// TIA Portal project "Esvetovaya" (V17)

(* hardware
DEVICE "S7-1200 station_1"  S7-1200 Station
   slot 0: "Rack_0"  S7-1200 Rack  Rack  V1.0
   slot 1: "PLC_1"  CPU 1214C AC/DC/Rly  6ES7 214-1BG40-0XB0  V4.5
*)

// ===== PLC "PLC_1"  CPU 1214C AC/DC/Rly =====

VAR_GLOBAL   // PLC tag table "TDB_Output_Q"
   "Q0.0_Lamp_Auto" AT %Q0.0 : Bool;   // Luces de modo automatico
   "Q0.1_Lamp_Manu" AT %Q0.1 : Bool;   // Luces de modo manual
   "Q0.2_Relay_ON" AT %Q0.2 : Bool;   // SAlida del soplador
   "Q0.3_Relay_ON" AT %Q0.3 : Bool;   // SAlida del soplador
   "Q0.4_Relay_ON" AT %Q0.4 : Bool;   // Salida de calefaccion
   "Q0.5_Relay_On" AT %Q0.5 : Bool;   // Salida de nebulizacion
   "Q1.0_Lamp_Auto_Running" AT %Q1.0 : Bool;   // Luces de modo de funcionamiento automatico
END_VAR

VAR_GLOBAL   // PLC tag table "TDB_Input_I"
   "I_Btt_Auto_Q0" AT %I0.0 : Bool;   // Modo de operacion Automatica
   "I_Btt_Manu_Q1" AT %I0.1 : Bool;   // Modo de operacion Manual
   "I_Btt_Start_Q2" AT %I0.2 : Bool;   // Interruptor de parada de funcionamiento del soplador
   "I_Btt___Off_Q2" AT %I0.3 : Bool;   // interruptor vegetariano deja de calentar
   "I_Btt_Start_Q3" AT %I0.4 : Bool;   // interruptor de funcionamiento detener nebulizacion
   "I_Btt___Off_Q3" AT %I0.5 : Bool;   // boton pulsador se ejecuta automaticamente
   "I_Btt_Start_Q4" AT %I0.6 : Bool;   // pulsador de parada automatica
   "Sensor_PT100" AT %IW64 : Int;   // sensor de temperatura
END_VAR

VAR_GLOBAL   // PLC tag table "M_Variables"
   "M_Btt_auto_Q0" AT %M0.0 : Bool;   // Memoria_Modo de operacion Automatica
   "M_Btt_Manu_Q1" AT %M0.1 : Bool;   // Memoria_Modo de operacion Manual
   "M_AUTO" AT %M0.2 : Bool;
   "M_MANUAL" AT %M0.3 : Bool;
   "M_Btt_Auto_On" AT %M0.4 : Bool;   // Memoria_boton pulsador se ejecuta automaticamente
   "M_Btt_Auto_Off" AT %M0.5 : Bool;   // Memoria_pulsador de parada automatica
   "ReStart" AT %M1.0 : Bool;
   "Bucle_Amarillo" AT %M1.1 : Bool;
   "Bucle_Rojo" AT %M1.3 : Bool;
   "M_SinEntender" AT %M1.4 : Bool;
   "M_Simulation" AT %M1.5 : Bool;   // Enciende la funciona de simulacion
   "Mtime_Lectura_Sensor" AT %M2.0 : Bool;
   "MQ2_Manu_Start" AT %M3.0 : Bool;   // Nebulizacion manual de modo intermedio
   "MQ2_Manu_Stop" AT %M3.1 : Bool;
   "MQ3_Manu_Start" AT %M3.2 : Bool;   // Soplador manual de modo intermedio
   "MQ3_Manu_Stop" AT %M3.3 : Bool;   // Calefaccion Manual de modo intermedio
   "MQ2_Auto_Start1" AT %M4.0 : Bool;   // Calentamiento Automatico en modo intermedio
   "MQ2_Auto_Start2" AT %M4.1 : Bool;   // Calentamiento Automatico en modo intermedio
   "MQ2_Auto_Start3" AT %M4.2 : Bool;   // Calentamiento Automatico en modo intermedio
   "MQ2_Auto_Stop" AT %M4.3 : Bool;
   "MQ2_Remote_Start" AT %M5.0 : Bool;   // Memoria_Interruptor de parada de funcionamiento del soplador
   "MQ3_Remote_Start" AT %M5.1 : Bool;   // Memoria_interruptor de funcionamiento detener nebulizacion
   "MQ2_Remote_Stop" AT %M5.2 : Bool;
   "MQ3_Remote_Stop" AT %M5.3 : Bool;
   "foco" AT %M6.0 : Bool;
END_VAR

DATA_BLOCK "DB_Sensors"   // DB1
{ S7_Optimized_Access := 'FALSE' }
VERSION : 0.1
   VAR
      Data_Norm_PT100 : Real;
      Data_Redondeo_PT100 : Real;
      Data_Scalado_PT100 : Real;
      Data_Evaluation_TempPT100 : Real := 25.0;
      Temp_Min : Real := 20.0;
      Temp_Max : Real := 27.0;
   END_VAR
BEGIN
END_DATA_BLOCK

DATA_BLOCK "DB_Clock"   // DB2
{ S7_Optimized_Access := 'TRUE' }
VERSION : 0.1
   VAR
      Fecha_hora_1_sistema : DTL := DTL#1970-01-01-00:00:00;
      Fecha_hora_2_sistema : DTL := DTL#1970-01-01-00:00:00;
      Fecha_hora_1_local : DTL := DTL#1970-01-01-00:00:00;
      Fecha_hora_2_local : DTL := DTL#1970-01-01-00:00:00;
      Ret_val_sistema_1 : Word := 16#0;
      Ret_val_sistema_2 : Word := 16#0;
      Ret_val_local_1 : Word := 16#0;
      Ret_val_local_2 : Word := 16#0;
      Hora_sistema_1 : Time_Of_Day := TOD#00:00:00;
      Hora_sistema_2 : Time_Of_Day := TOD#00:00:00;
      Hora_local_1 : Time_Of_Day := TOD#00:00:00;
      Hora_local_2 : Time_Of_Day := TOD#00:00:00;
      Hora_Q2_inicio_1 : Time_Of_Day := TOD#00:00:00;
      Hora_Q2_inicio_2 : Time_Of_Day := TOD#00:00:00;
      Hora_Q2_inicio_3 : Time_Of_Day := TOD#00:00:00;
      Hora_Q3_inicio_1 : Time_Of_Day := TOD#00:00:00;
      Hora_Q3_inicio_2 : Time_Of_Day := TOD#00:00:00;
      Hora_Q3_inicio_3 : Time_Of_Day := TOD#00:00:00;
      Hora_Q2_fin_1 : Time_Of_Day := TOD#00:00:00;
      Hora_Q2_fin_2 : Time_Of_Day := TOD#00:00:00;
      Hora_Q2_fin_3 : Time_Of_Day := TOD#00:00:00;
      Hora_Q3_fin_1 : Time_Of_Day := TOD#00:00:00;
      Hora_Q3_fin_2 : Time_Of_Day := TOD#00:00:00;
      Hora_Q3_fin_3 : Time_Of_Day := TOD#00:00:00;
      Hora_Start_ARR_Q2_1 : Array[1..7] of Time_Of_Day;
      Hora_Start_ARR_Q2_2 : Array[1..7] of Time_Of_Day;
      Hora_Start_ARR_Q2_3 : Array[1..7] of Time_Of_Day;
      Hora_Start_ARR_Q3_1 : Array[1..7] of Time_Of_Day;
      Hora_Start_ARR_Q3_2 : Array[1..7] of Time_Of_Day;
      Hora_Start_ARR_Q3_3 : Array[1..7] of Time_Of_Day;
      Hora_End_ARR_Q2_1 : Array[1..7] of Time_Of_Day;
      Hora_End_ARR_Q2_2 : Array[1..7] of Time_Of_Day;
      Hora_End_ARR_Q2_3 : Array[1..7] of Time_Of_Day;
      Hora_End_ARR_Q3_1 : Array[1..7] of Time_Of_Day;
      Hora_End_ARR_Q3_2 : Array[1..7] of Time_Of_Day;
      Hora_End_ARR_Q3_3 : Array[1..7] of Time_Of_Day;
   END_VAR
BEGIN
   Hora_Start_ARR_Q2_1[1] := TOD#06:00:00;
   Hora_Start_ARR_Q2_1[2] := TOD#06:00:00;
   Hora_Start_ARR_Q2_1[3] := TOD#06:00:00;
   Hora_Start_ARR_Q2_1[4] := TOD#06:00:00;
   Hora_Start_ARR_Q2_1[5] := TOD#06:00:00;
   Hora_Start_ARR_Q2_1[6] := TOD#06:00:00;
   Hora_Start_ARR_Q2_1[7] := TOD#06:00:00;
   Hora_End_ARR_Q2_1[1] := TOD#20:00:00;
   Hora_End_ARR_Q2_1[2] := TOD#20:00:00;
   Hora_End_ARR_Q2_1[3] := TOD#20:00:00;
   Hora_End_ARR_Q2_1[4] := TOD#20:00:00;
   Hora_End_ARR_Q2_1[5] := TOD#20:00:00;
   Hora_End_ARR_Q2_1[6] := TOD#20:00:00;
   Hora_End_ARR_Q2_1[7] := TOD#20:00:00;
   Hora_Start_ARR_Q2_2[1] := TOD#06:00:00;
   Hora_Start_ARR_Q2_2[2] := TOD#06:00:00;
   Hora_Start_ARR_Q2_2[3] := TOD#06:00:00;
   Hora_Start_ARR_Q2_2[4] := TOD#06:00:00;
   Hora_Start_ARR_Q2_2[5] := TOD#06:00:00;
   Hora_Start_ARR_Q2_2[6] := TOD#06:00:00;
   Hora_Start_ARR_Q2_2[7] := TOD#06:00:00;
   Hora_Start_ARR_Q2_3[1] := TOD#06:00:00;
   Hora_Start_ARR_Q2_3[2] := TOD#06:00:00;
   Hora_Start_ARR_Q2_3[3] := TOD#06:00:00;
   Hora_Start_ARR_Q2_3[4] := TOD#06:00:00;
   Hora_Start_ARR_Q2_3[5] := TOD#06:00:00;
   Hora_Start_ARR_Q2_3[6] := TOD#06:00:00;
   Hora_Start_ARR_Q2_3[7] := TOD#06:00:00;
   Hora_Start_ARR_Q3_1[1] := TOD#06:00:00;
   Hora_Start_ARR_Q3_1[2] := TOD#06:00:00;
   Hora_Start_ARR_Q3_1[3] := TOD#06:00:00;
   Hora_Start_ARR_Q3_1[4] := TOD#06:00:00;
   Hora_Start_ARR_Q3_1[5] := TOD#06:00:00;
   Hora_Start_ARR_Q3_1[6] := TOD#06:00:00;
   Hora_Start_ARR_Q3_1[7] := TOD#06:00:00;
   Hora_Start_ARR_Q3_2[1] := TOD#06:00:00;
   Hora_Start_ARR_Q3_2[2] := TOD#06:00:00;
   Hora_Start_ARR_Q3_2[3] := TOD#06:00:00;
   Hora_Start_ARR_Q3_2[4] := TOD#06:00:00;
   Hora_Start_ARR_Q3_2[5] := TOD#06:00:00;
   Hora_Start_ARR_Q3_2[6] := TOD#06:00:00;
   Hora_Start_ARR_Q3_2[7] := TOD#06:00:00;
   Hora_Start_ARR_Q3_3[1] := TOD#06:00:00;
   Hora_Start_ARR_Q3_3[2] := TOD#06:00:00;
   Hora_Start_ARR_Q3_3[3] := TOD#06:00:00;
   Hora_Start_ARR_Q3_3[4] := TOD#06:00:00;
   Hora_Start_ARR_Q3_3[5] := TOD#06:00:00;
   Hora_Start_ARR_Q3_3[6] := TOD#06:00:00;
   Hora_Start_ARR_Q3_3[7] := TOD#06:00:00;
   Hora_End_ARR_Q2_2[1] := TOD#20:00:00;
   Hora_End_ARR_Q2_2[2] := TOD#20:00:00;
   Hora_End_ARR_Q2_2[3] := TOD#20:00:00;
   Hora_End_ARR_Q2_2[4] := TOD#20:00:00;
   Hora_End_ARR_Q2_2[5] := TOD#20:00:00;
   Hora_End_ARR_Q2_2[6] := TOD#20:00:00;
   Hora_End_ARR_Q2_2[7] := TOD#20:00:00;
   Hora_End_ARR_Q2_3[1] := TOD#20:00:00;
   Hora_End_ARR_Q2_3[2] := TOD#20:00:00;
   Hora_End_ARR_Q2_3[3] := TOD#20:00:00;
   Hora_End_ARR_Q2_3[4] := TOD#20:00:00;
   Hora_End_ARR_Q2_3[5] := TOD#20:00:00;
   Hora_End_ARR_Q2_3[6] := TOD#20:00:00;
   Hora_End_ARR_Q2_3[7] := TOD#20:00:00;
   Hora_End_ARR_Q3_1[1] := TOD#20:00:00;
   Hora_End_ARR_Q3_1[2] := TOD#20:00:00;
   Hora_End_ARR_Q3_1[3] := TOD#20:00:00;
   Hora_End_ARR_Q3_1[4] := TOD#20:00:00;
   Hora_End_ARR_Q3_1[5] := TOD#20:00:00;
   Hora_End_ARR_Q3_1[6] := TOD#20:00:00;
   Hora_End_ARR_Q3_1[7] := TOD#20:00:00;
   Hora_End_ARR_Q3_2[1] := TOD#20:00:00;
   Hora_End_ARR_Q3_2[2] := TOD#20:00:00;
   Hora_End_ARR_Q3_2[3] := TOD#20:00:00;
   Hora_End_ARR_Q3_2[4] := TOD#20:00:00;
   Hora_End_ARR_Q3_2[5] := TOD#20:00:00;
   Hora_End_ARR_Q3_2[6] := TOD#20:00:00;
   Hora_End_ARR_Q3_2[7] := TOD#20:00:00;
   Hora_End_ARR_Q3_3[1] := TOD#20:00:00;
   Hora_End_ARR_Q3_3[2] := TOD#20:00:00;
   Hora_End_ARR_Q3_3[3] := TOD#20:00:00;
   Hora_End_ARR_Q3_3[4] := TOD#20:00:00;
   Hora_End_ARR_Q3_3[5] := TOD#20:00:00;
   Hora_End_ARR_Q3_3[6] := TOD#20:00:00;
   Hora_End_ARR_Q3_3[7] := TOD#20:00:00;
END_DATA_BLOCK

DATA_BLOCK "DB_Retain"   // DB3
{ S7_Optimized_Access := 'TRUE' }
VERSION : 0.1
   VAR RETAIN
      M_Btt_auto : Bool;
   END_VAR
BEGIN
END_DATA_BLOCK

DATA_BLOCK "Datos"   // DB7
{ S7_Optimized_Access := 'FALSE' }
VERSION : 0.1
   VAR
      Static_1 : Bool;
      DatoEntero : Array[0..4] of Int;
      DatoReal : Array[0..4] of Real;
      DatoWord : Array[0..4] of Word;
      DatoBooleano : Array[0..4] of Bool;
   END_VAR
BEGIN
END_DATA_BLOCK

DATA_BLOCK "DB_Input"   // DB8
{ S7_Optimized_Access := 'TRUE' }
VERSION : 0.1
   VAR
      "1" : Bool;
   END_VAR
BEGIN
END_DATA_BLOCK

// folder: System blocks/Program resources

DATA_BLOCK "IEC_Timer_0_DB"   // DB4
{ S7_Optimized_Access := 'TRUE' }
AUTHOR : Simatic
FAMILY : IEC
NAME : IEC_TMR
VERSION : 1.0
// stored: InstanceOfName IEC_TIMER
"IEC_TIMER"
BEGIN
END_DATA_BLOCK

DATA_BLOCK "IEC_Timer_0_DB_1"   // DB5
{ S7_Optimized_Access := 'TRUE' }
AUTHOR : Simatic
FAMILY : IEC
NAME : IEC_TMR
VERSION : 1.0
// stored: InstanceOfName IEC_TIMER
"IEC_TIMER"
BEGIN
END_DATA_BLOCK

DATA_BLOCK "IEC_Timer_0_DB_2"   // DB6
{ S7_Optimized_Access := 'TRUE' }
AUTHOR : Simatic
FAMILY : IEC
NAME : IEC_TMR
VERSION : 1.0
// stored: InstanceOfName IEC_TIMER
"IEC_TIMER"
BEGIN
END_DATA_BLOCK

// folder: (top level)

FUNCTION "FC_MANUAL" : Void   // FC1, LAD
{ S7_Optimized_Access := 'TRUE' }
VERSION : 0.1
BEGIN

REGION Network 1: выход Q2 - MANUAL-(ON-OFF)
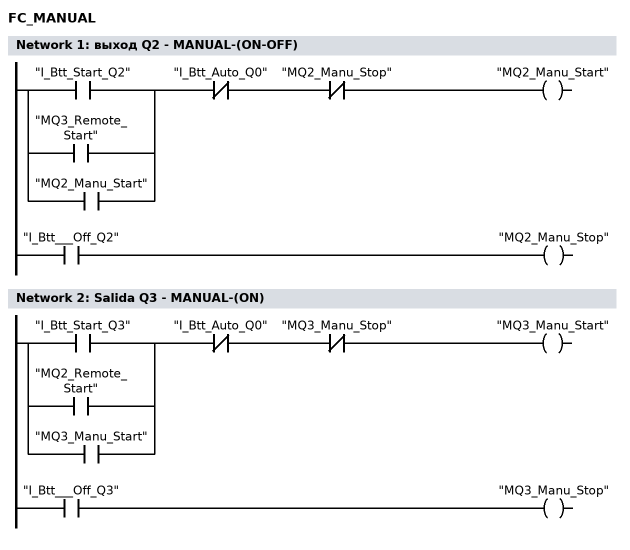
   RUNG wire#powerrail
      Contact( "I_Btt_Start_Q2" )
      wire#w1
      I_Contact( "I_Btt_Auto_Q0" )
      I_Contact( "MQ2_Manu_Stop" )
      Coil( "MQ2_Manu_Start" )
   END_RUNG
   RUNG wire#powerrail
      Contact( "MQ3_Remote_Start" )
   END_RUNG wire#w1
   RUNG wire#powerrail
      Contact( "MQ2_Manu_Start" )
   END_RUNG wire#w1
   RUNG wire#powerrail
      Contact( "I_Btt___Off_Q2" )
      Coil( "MQ2_Manu_Stop" )
   END_RUNG
   // the same network as SCL:
   "MQ2_Manu_Start" := ("I_Btt_Start_Q2" OR "MQ3_Remote_Start" OR "MQ2_Manu_Start") AND NOT "I_Btt_Auto_Q0" AND NOT "MQ2_Manu_Stop";
   "MQ2_Manu_Stop" := "I_Btt___Off_Q2";
END_REGION

REGION Network 2: Salida Q3 - MANUAL-(ON)
   RUNG wire#powerrail
      Contact( "I_Btt_Start_Q3" )
      wire#w1
      I_Contact( "I_Btt_Auto_Q0" )
      I_Contact( "MQ3_Manu_Stop" )
      Coil( "MQ3_Manu_Start" )
   END_RUNG
   RUNG wire#powerrail
      Contact( "MQ2_Remote_Start" )
   END_RUNG wire#w1
   RUNG wire#powerrail
      Contact( "MQ3_Manu_Start" )
   END_RUNG wire#w1
   RUNG wire#powerrail
      Contact( "I_Btt___Off_Q3" )
      Coil( "MQ3_Manu_Stop" )
   END_RUNG
   // the same network as SCL:
   "MQ3_Manu_Start" := ("I_Btt_Start_Q3" OR "MQ2_Remote_Start" OR "MQ3_Manu_Start") AND NOT "I_Btt_Auto_Q0" AND NOT "MQ3_Manu_Stop";
   "MQ3_Manu_Stop" := "I_Btt___Off_Q3";
END_REGION
END_FUNCTION

FUNCTION "FC_AUTO" : Void   // FC2, LAD
{ S7_Optimized_Access := 'TRUE' }
VERSION : 0.1
BEGIN

REGION Network 1: Memoria REINICIO PLC-AUTOMATICO
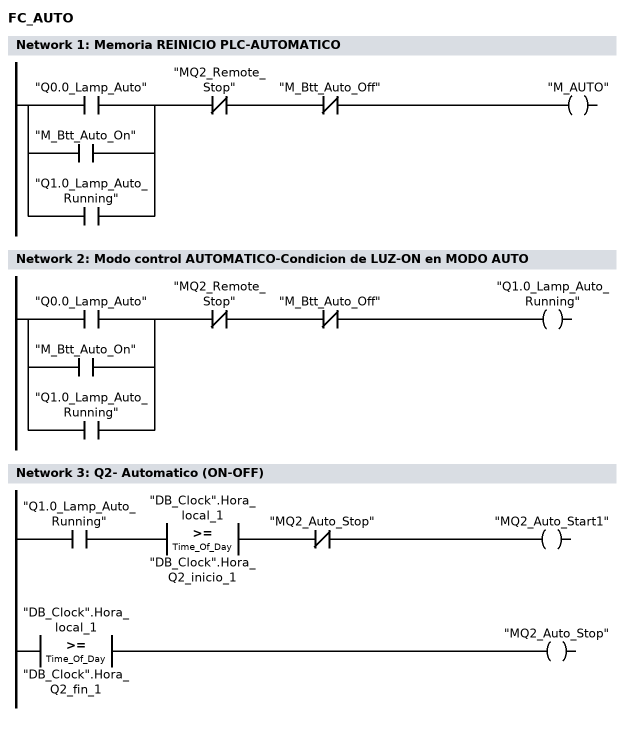
   RUNG wire#powerrail
      Contact( "Q0.0_Lamp_Auto" )
      wire#w1
      I_Contact( "MQ2_Remote_Stop" )
      I_Contact( "M_Btt_Auto_Off" )
      Coil( "M_AUTO" )
   END_RUNG
   RUNG wire#powerrail
      Contact( "M_Btt_Auto_On" )
   END_RUNG wire#w1
   RUNG wire#powerrail
      Contact( "Q1.0_Lamp_Auto_Running" )
   END_RUNG wire#w1
   // the same network as SCL:
   "M_AUTO" := ("Q0.0_Lamp_Auto" OR "M_Btt_Auto_On" OR "Q1.0_Lamp_Auto_Running") AND NOT "MQ2_Remote_Stop" AND NOT "M_Btt_Auto_Off";
END_REGION

REGION Network 2: Modo control AUTOMATICO-Condicion de LUZ-ON en MODO AUTO
   RUNG wire#powerrail
      Contact( "Q0.0_Lamp_Auto" )
      wire#w1
      I_Contact( "MQ2_Remote_Stop" )
      I_Contact( "M_Btt_Auto_Off" )
      Coil( "Q1.0_Lamp_Auto_Running" )
   END_RUNG
   RUNG wire#powerrail
      Contact( "M_Btt_Auto_On" )
   END_RUNG wire#w1
   RUNG wire#powerrail
      Contact( "Q1.0_Lamp_Auto_Running" )
   END_RUNG wire#w1
   // the same network as SCL:
   "Q1.0_Lamp_Auto_Running" := ("Q0.0_Lamp_Auto" OR "M_Btt_Auto_On" OR "Q1.0_Lamp_Auto_Running") AND NOT "MQ2_Remote_Stop" AND NOT "M_Btt_Auto_Off";
END_REGION

REGION Network 3: Q2- Automatico (ON-OFF)
   RUNG wire#powerrail
      Contact( "Q1.0_Lamp_Auto_Running" )
      { S7_Templates := "SrcType := Time_Of_Day" } GE_Contact(in1 := "DB_Clock".Hora_local_1, in2 := "DB_Clock".Hora_Q2_inicio_1)
      I_Contact( "MQ2_Auto_Stop" )
      Coil( "MQ2_Auto_Start1" )
   END_RUNG
   RUNG wire#powerrail
      { S7_Templates := "SrcType := Time_Of_Day" } GE_Contact(in1 := "DB_Clock".Hora_local_1, in2 := "DB_Clock".Hora_Q2_fin_1)
      Coil( "MQ2_Auto_Stop" )
   END_RUNG
   // the same network as SCL:
   "MQ2_Auto_Start1" := "Q1.0_Lamp_Auto_Running" AND ("DB_Clock".Hora_local_1 >= "DB_Clock".Hora_Q2_inicio_1) AND NOT "MQ2_Auto_Stop";
   "MQ2_Auto_Stop" := "DB_Clock".Hora_local_1 >= "DB_Clock".Hora_Q2_fin_1;
END_REGION
END_FUNCTION

FUNCTION "FC_OUTPUT_Q" : Void   // FC3, LAD
{ S7_Optimized_Access := 'TRUE' }
VERSION : 0.1
BEGIN

REGION Network 1: Salida Q-02 (On-Off)
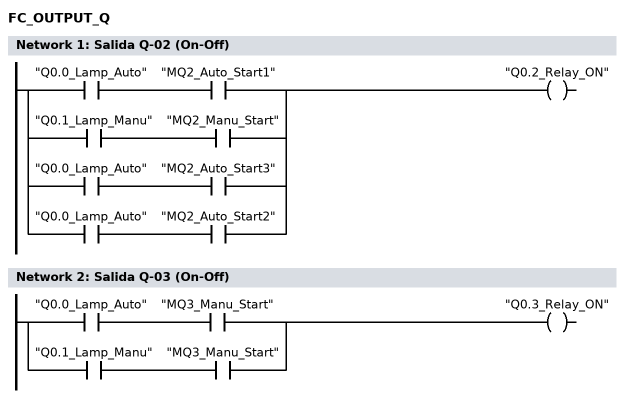
   RUNG wire#powerrail
      Contact( "Q0.0_Lamp_Auto" )
      Contact( "MQ2_Auto_Start1" )
      wire#w1
      Coil( "Q0.2_Relay_ON" )
   END_RUNG
   RUNG wire#powerrail
      Contact( "Q0.1_Lamp_Manu" )
      Contact( "MQ2_Manu_Start" )
   END_RUNG wire#w1
   RUNG wire#powerrail
      Contact( "Q0.0_Lamp_Auto" )
      Contact( "MQ2_Auto_Start3" )
   END_RUNG wire#w1
   RUNG wire#powerrail
      Contact( "Q0.0_Lamp_Auto" )
      Contact( "MQ2_Auto_Start2" )
   END_RUNG wire#w1
   // the same network as SCL:
   "Q0.2_Relay_ON" := ("Q0.0_Lamp_Auto" AND "MQ2_Auto_Start1") OR ("Q0.1_Lamp_Manu" AND "MQ2_Manu_Start") OR ("Q0.0_Lamp_Auto" AND "MQ2_Auto_Start3") OR ("Q0.0_Lamp_Auto" AND "MQ2_Auto_Start2");
END_REGION

REGION Network 2: Salida Q-03 (On-Off)
   RUNG wire#powerrail
      Contact( "Q0.0_Lamp_Auto" )
      Contact( "MQ3_Manu_Start" )
      wire#w1
      Coil( "Q0.3_Relay_ON" )
   END_RUNG
   RUNG wire#powerrail
      Contact( "Q0.1_Lamp_Manu" )
      Contact( "MQ3_Manu_Start" )
   END_RUNG wire#w1
   // the same network as SCL:
   "Q0.3_Relay_ON" := ("Q0.0_Lamp_Auto" AND "MQ3_Manu_Start") OR ("Q0.1_Lamp_Manu" AND "MQ3_Manu_Start");
END_REGION
END_FUNCTION

FUNCTION "FC_SENSORS" : Void   // FC4, LAD
{ S7_Optimized_Access := 'TRUE' }
VERSION : 0.1
BEGIN

REGION Network 1
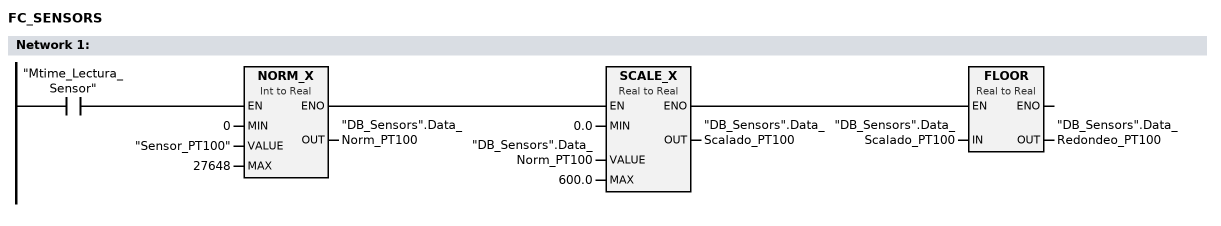
   IF "Mtime_Lectura_Sensor" THEN
       "DB_Sensors".Data_Norm_PT100 := NORM_X(MIN := 0, VALUE := "Sensor_PT100", MAX := 27648);
       "DB_Sensors".Data_Scalado_PT100 := SCALE_X(MIN := 0.0, VALUE := "DB_Sensors".Data_Norm_PT100, MAX := 600.0);
       "DB_Sensors".Data_Redondeo_PT100 := FLOOR("DB_Sensors".Data_Scalado_PT100);
   END_IF;
END_REGION
END_FUNCTION

FUNCTION "FC_CLOCK" : Void   // FC5, LAD
{ S7_Optimized_Access := 'TRUE' }
VERSION : 0.1
BEGIN

REGION Network 1: Tiempo de INTERVALO DE LECTURA FC_SENSORS
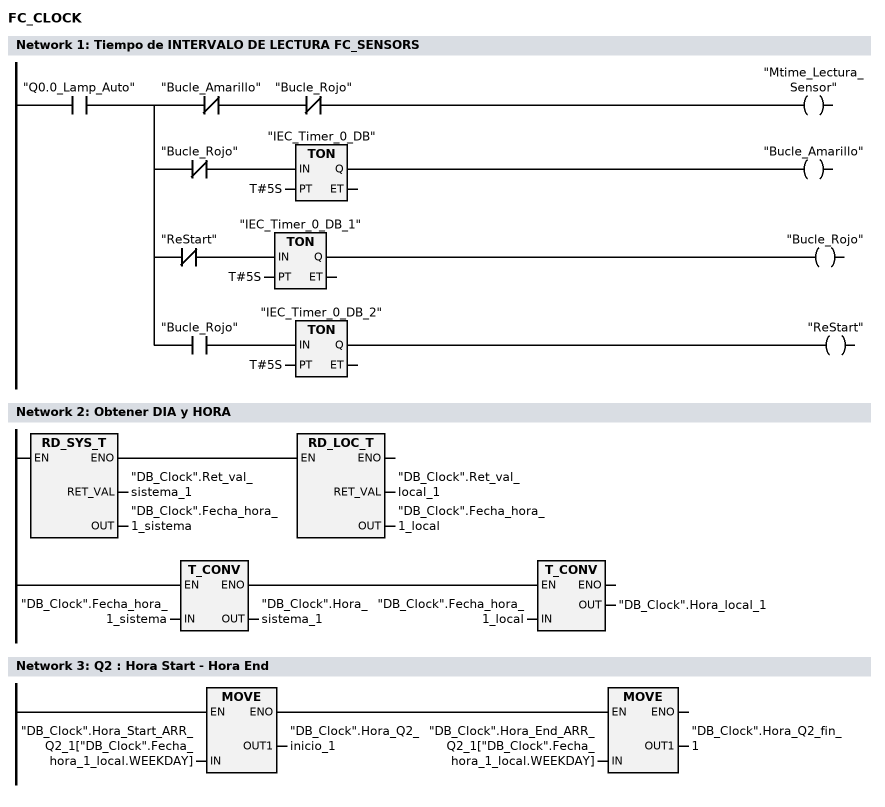
   "Mtime_Lectura_Sensor" := "Q0.0_Lamp_Auto" AND NOT "Bucle_Amarillo" AND NOT "Bucle_Rojo";
   "IEC_Timer_0_DB".TON(IN := "Q0.0_Lamp_Auto" AND NOT "Bucle_Rojo", PT := T#5S);
   "Bucle_Amarillo" := "IEC_Timer_0_DB".Q;
   "IEC_Timer_0_DB_1".TON(IN := "Q0.0_Lamp_Auto" AND NOT "ReStart", PT := T#5S);
   "Bucle_Rojo" := "IEC_Timer_0_DB_1".Q;
   "IEC_Timer_0_DB_2".TON(IN := "Q0.0_Lamp_Auto" AND "Bucle_Rojo", PT := T#5S);
   "ReStart" := "IEC_Timer_0_DB_2".Q;
END_REGION

REGION Network 2: Obtener DIA y HORA
   // ENO of a box is taken as its EN; it also drops when the box reports an error
   "DB_Clock".Ret_val_sistema_1 := RD_SYS_T(OUT => "DB_Clock".Fecha_hora_1_sistema);
   "DB_Clock".Ret_val_local_1 := RD_LOC_T(OUT => "DB_Clock".Fecha_hora_1_local);
   "DB_Clock".Hora_sistema_1 := T_CONV(IN := "DB_Clock".Fecha_hora_1_sistema);
   "DB_Clock".Hora_local_1 := T_CONV(IN := "DB_Clock".Fecha_hora_1_local);
END_REGION

REGION Network 3: Q2 : Hora Start - Hora End
   RUNG wire#powerrail
      Move(in := "DB_Clock".Hora_Start_ARR_Q2_1["DB_Clock".Fecha_hora_1_local.WEEKDAY], out1 => "DB_Clock".Hora_Q2_inicio_1)
      Move(in := "DB_Clock".Hora_End_ARR_Q2_1["DB_Clock".Fecha_hora_1_local.WEEKDAY], out1 => "DB_Clock".Hora_Q2_fin_1)
   END_RUNG
   // the same network as SCL:
   "DB_Clock".Hora_Q2_inicio_1 := "DB_Clock".Hora_Start_ARR_Q2_1["DB_Clock".Fecha_hora_1_local.WEEKDAY];
   "DB_Clock".Hora_Q2_fin_1 := "DB_Clock".Hora_End_ARR_Q2_1["DB_Clock".Fecha_hora_1_local.WEEKDAY];
END_REGION
END_FUNCTION

ORGANIZATION_BLOCK "Main"   // OB1, LAD, ProgramCycle
TITLE = "Main Program Sweep (Cycle)"
{ S7_Optimized_Access := 'TRUE' }
VERSION : 0.1
   VAR_INPUT
      Initial_Call : Bool;   // Initial call of this OB
      Remanence : Bool;   // =True, if remanent data are available
   END_VAR
   VAR_TEMP   // added for the SCL form of the ladder/FBD networks
      _w1 : Bool;
   END_VAR
BEGIN

REGION Network 1: Programa AUTOMATICO
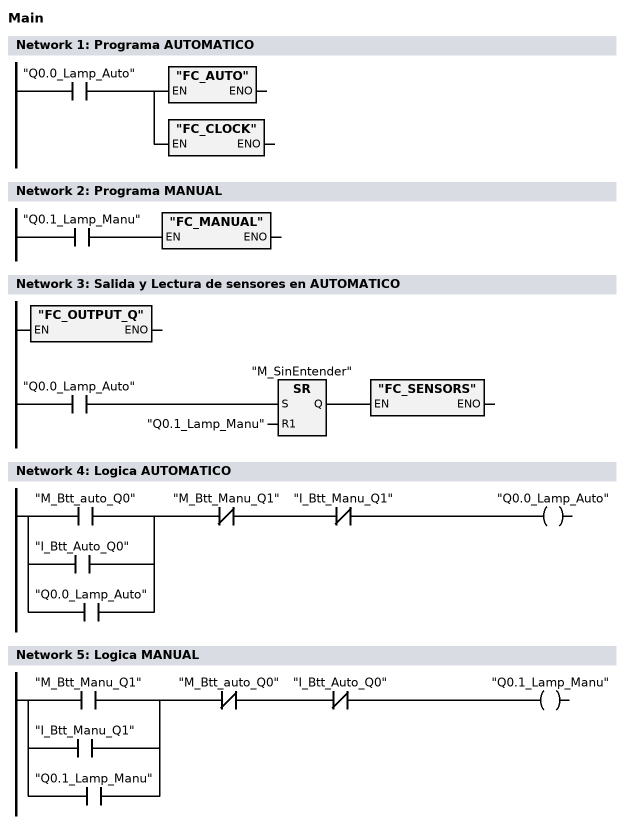
   RUNG wire#powerrail
      Contact( "Q0.0_Lamp_Auto" )
      wire#w1
      "FC_AUTO"()
   END_RUNG
   RUNG wire#w1
      "FC_CLOCK"()
   END_RUNG
   // the same network as SCL:
   #_w1 := "Q0.0_Lamp_Auto";
   IF #_w1 THEN
       "FC_AUTO"();
       "FC_CLOCK"();
   END_IF;
END_REGION

REGION Network 2: Programa MANUAL
   RUNG wire#powerrail
      Contact( "Q0.1_Lamp_Manu" )
      "FC_MANUAL"()
   END_RUNG
   // the same network as SCL:
   IF "Q0.1_Lamp_Manu" THEN "FC_MANUAL"(); END_IF;
END_REGION

REGION Network 3: Salida y Lectura de sensores en AUTOMATICO
   RUNG wire#powerrail
      "FC_OUTPUT_Q"()
   END_RUNG
   RUNG wire#powerrail
      Contact( "Q0.0_Lamp_Auto" )
      S_SR(operand := "M_SinEntender", r1 := "Q0.1_Lamp_Manu")
      "FC_SENSORS"()
   END_RUNG
   // the same network as SCL:
   "FC_OUTPUT_Q"();
   IF "Q0.0_Lamp_Auto" THEN
       "M_SinEntender" := TRUE;   // SR flip-flop
   END_IF;
   IF "Q0.1_Lamp_Manu" THEN "M_SinEntender" := FALSE; END_IF;
   IF "M_SinEntender" THEN "FC_SENSORS"(); END_IF;
END_REGION

REGION Network 4: Logica AUTOMATICO
   RUNG wire#powerrail
      Contact( "M_Btt_auto_Q0" )
      wire#w1
      I_Contact( "M_Btt_Manu_Q1" )
      I_Contact( "I_Btt_Manu_Q1" )
      Coil( "Q0.0_Lamp_Auto" )
   END_RUNG
   RUNG wire#powerrail
      Contact( "I_Btt_Auto_Q0" )
   END_RUNG wire#w1
   RUNG wire#powerrail
      Contact( "Q0.0_Lamp_Auto" )
   END_RUNG wire#w1
   // the same network as SCL:
   "Q0.0_Lamp_Auto" := ("M_Btt_auto_Q0" OR "I_Btt_Auto_Q0" OR "Q0.0_Lamp_Auto") AND NOT "M_Btt_Manu_Q1" AND NOT "I_Btt_Manu_Q1";
END_REGION

REGION Network 5: Logica MANUAL
   RUNG wire#powerrail
      Contact( "M_Btt_Manu_Q1" )
      wire#w1
      I_Contact( "M_Btt_auto_Q0" )
      I_Contact( "I_Btt_Auto_Q0" )
      Coil( "Q0.1_Lamp_Manu" )
   END_RUNG
   RUNG wire#powerrail
      Contact( "I_Btt_Manu_Q1" )
   END_RUNG wire#w1
   RUNG wire#powerrail
      Contact( "Q0.1_Lamp_Manu" )
   END_RUNG wire#w1
   // the same network as SCL:
   "Q0.1_Lamp_Manu" := ("M_Btt_Manu_Q1" OR "I_Btt_Manu_Q1" OR "Q0.1_Lamp_Manu") AND NOT "M_Btt_auto_Q0" AND NOT "I_Btt_Auto_Q0";
END_REGION
END_ORGANIZATION_BLOCK

ORGANIZATION_BLOCK "Startup"   // OB100, LAD, Startup
TITLE = "Complete Restart"
{ S7_Optimized_Access := 'TRUE' }
VERSION : 0.1
   VAR_INPUT
      LostRetentive : Bool;   // True if retentive data are lost
      LostRTC : Bool;   // True if date and time are lost
   END_VAR
BEGIN

REGION Network 1: Luces de modo automatico
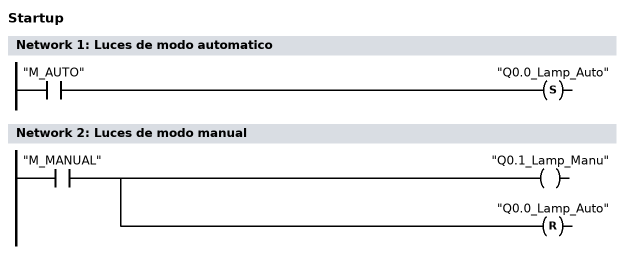
   RUNG wire#powerrail
      Contact( "M_AUTO" )
      S_Coil( "Q0.0_Lamp_Auto" )
   END_RUNG
   // the same network as SCL:
   IF "M_AUTO" THEN "Q0.0_Lamp_Auto" := TRUE; END_IF;
END_REGION

REGION Network 2: Luces de modo manual
   RUNG wire#powerrail
      Contact( "M_MANUAL" )
      wire#w1
      Coil( "Q0.1_Lamp_Manu" )
   END_RUNG
   RUNG wire#w1
      R_Coil( "Q0.0_Lamp_Auto" )
   END_RUNG
   // the same network as SCL:
   "Q0.1_Lamp_Manu" := "M_MANUAL";
   IF "M_MANUAL" THEN "Q0.0_Lamp_Auto" := FALSE; END_IF;
END_REGION
END_ORGANIZATION_BLOCK